(* IEC 61131-3 sources: Word/plc-course/05-boolean-logic-and-fbd/labs/solutions, 3 files *)

(* ---- 05-1-pump-permissive.st ---- *)
(* Lab 05-1: Transfer pump P-101 start permissive.
   Module 05 (Boolean logic and FBD). REFERENCE SOLUTION - try the lab yourself first.

   Everything here is combinational: every output depends only on the inputs
   of the present scan. There is no seal-in, latch or timer. *)

PROGRAM TransferPump
  VAR (* I/O - addresses follow the OpenPLC convention *)
    SuctionOpenLS AT %IX0.0 : BOOL;  (* Suction valve XV-100 open limit switch (ZSO-100): TRUE = fully open *)
    LSL101_NC     AT %IX0.1 : BOOL;  (* Tank low-level switch LSL-101, NC: TRUE = level above the switch (healthy) *)
    MotorFault    AT %IX0.2 : BOOL;  (* Motor protection relay fault contact, NO: TRUE = protection tripped *)
    ManualSel     AT %IX0.3 : BOOL;  (* MAN-OFF-AUTO selector, MAN contact *)
    AutoSel       AT %IX0.4 : BOOL;  (* MAN-OFF-AUTO selector, AUTO contact *)
    Demand        AT %IX0.5 : BOOL;  (* Auto demand from the process: TRUE = liquid wanted *)
    ManualRunCmd  AT %IX0.6 : BOOL;  (* Manual run command, maintained: TRUE = run *)
    Pump          AT %QX0.0 : BOOL;  (* P-101 motor starter: TRUE = run *)
    PermissiveOK  AT %QX0.1 : BOOL;  (* White "Ready" lamp: all start permissives healthy *)
    SelectorFault AT %QX0.2 : BOOL;  (* Both selector contacts made at once *)
  END_VAR
  VAR (* internal *)
    AutoMode   : BOOL;  (* selector cleanly in AUTO *)
    ManualMode : BOOL;  (* selector cleanly in MAN *)
    RunRequest : BOOL;  (* the active mode is asking for the pump *)
  END_VAR

  (* 1. Permissives. Each input is used in the sense that means "healthy":
        LSL101_NC is wired fail-safe and is already TRUE when healthy, so it is
        used as it is. MotorFault is TRUE when faulted, so it needs a NOT. *)
  PermissiveOK := SuctionOpenLS AND LSL101_NC AND NOT MotorFault;

  (* 2. Mode. A healthy three-position selector closes at most one contact.
        Both contacts at once is a fault, and it must not select any mode. *)
  SelectorFault := ManualSel AND AutoSel;
  AutoMode      := AutoSel AND NOT ManualSel;
  ManualMode    := ManualSel AND NOT AutoSel;

  (* 3. What the active mode asks for. The parentheses are not strictly needed
        (AND binds tighter than OR), but they show the intent at a glance. *)
  RunRequest := (AutoMode AND Demand) OR (ManualMode AND ManualRunCmd);

  (* 4. The permissives apply in every mode, so they go outside the OR. *)
  Pump := PermissiveOK AND RunRequest;
END_PROGRAM

CONFIGURATION Config0
  RESOURCE Res0 ON PLC
    TASK MainTask(INTERVAL := T#10ms, PRIORITY := 0);
    PROGRAM Inst0 WITH MainTask : TransferPump;
  END_RESOURCE
END_CONFIGURATION

(* ---- 05-2-two-out-of-three-vote.st ---- *)
(* Lab 05-2: Two-out-of-three (2oo3) high-pressure trip vote.
   Module 05 (Boolean logic and FBD). REFERENCE SOLUTION - try the lab yourself first.

   TRAINING EXERCISE ONLY. This shows the Boolean logic of voting. It is not a
   design for a real safety function: real trips run in a safety-rated system
   engineered to IEC 61511 / IEC 61508 (Module 20), and they latch until reset. *)

PROGRAM TripVote
  VAR (* I/O - addresses follow the OpenPLC convention *)
    PSHH_A_NC   AT %IX0.0 : BOOL;  (* PSHH-101A, NC: TRUE = pressure below trip setting (healthy) *)
    PSHH_B_NC   AT %IX0.1 : BOOL;  (* PSHH-101B, NC: as above *)
    PSHH_C_NC   AT %IX0.2 : BOOL;  (* PSHH-101C, NC: as above *)
    Trip        AT %QX0.0 : BOOL;  (* TRUE = at least two channels demand a trip *)
    SDVSolenoid AT %QX0.1 : BOOL;  (* SDV-100 solenoid: TRUE = energised, valve held open *)
    Discrepancy AT %QX0.2 : BOOL;  (* TRUE = the three channels do not all agree *)
    DiscA       AT %QX0.3 : BOOL;  (* TRUE = channel A disagrees with B and C *)
    DiscB       AT %QX0.4 : BOOL;  (* TRUE = channel B disagrees with A and C *)
    DiscC       AT %QX0.5 : BOOL;  (* TRUE = channel C disagrees with A and B *)
  END_VAR
  VAR (* internal: channel trip demands, TRUE = this channel says "trip" *)
    DemA : BOOL;
    DemB : BOOL;
    DemC : BOOL;
  END_VAR

  (* 1. Convert each fail-safe input into "this channel demands a trip".
        High pressure opens the contact, and so does a broken wire: both
        read FALSE, and both count as a demand. *)
  DemA := NOT PSHH_A_NC;
  DemB := NOT PSHH_B_NC;
  DemC := NOT PSHH_C_NC;

  (* 2. Majority vote: any two of the three. *)
  Trip := (DemA AND DemB) OR (DemB AND DemC) OR (DemA AND DemC);

  (* 3. De-energise to trip: the solenoid is powered only while there is no trip. *)
  SDVSolenoid := NOT Trip;

  (* 4. Which channel is the odd one out? A channel disagrees with the others
        when it differs from BOTH of them (which also means the other two agree). *)
  DiscA := (DemA XOR DemB) AND (DemA XOR DemC);
  DiscB := (DemB XOR DemA) AND (DemB XOR DemC);
  DiscC := (DemC XOR DemA) AND (DemC XOR DemB);

  (* 5. With three two-state channels, "not all equal" always means exactly
        one channel is the odd one out, so this is the same as
        (DemA XOR DemB) OR (DemB XOR DemC). *)
  Discrepancy := DiscA OR DiscB OR DiscC;
END_PROGRAM

CONFIGURATION Config0
  RESOURCE Res0 ON PLC
    TASK MainTask(INTERVAL := T#10ms, PRIORITY := 0);
    PROGRAM Inst0 WITH MainTask : TripVote;
  END_RESOURCE
END_CONFIGURATION

(* ---- 05-3-horn-truth-table.st ---- *)
(* Lab 05-3: From truth table to minimal logic - wet-well alarm horn.
   Module 05 (Boolean logic and FBD). REFERENCE SOLUTION - try the lab yourself first.

   K-map (rows HighLevel LowLevel, columns Pump1Run Pump2Run, Gray order):

                    P1 P2:  00   01   11   10
     H L = 00               0    0    0    0
     H L = 01               0    1    1    1
     H L = 11               1    1    1    1
     H L = 10               1    0    0    0

   Groups:  L.P2      quad  (rows 01, 11 x columns 01, 11)
            L.P1      quad  (rows 01, 11 x columns 11, 10)
            H.P1'.P2' pair  (rows 11, 10 x column 00)
   Every group is essential, so the minimal sum of products is unique:
     Horn = L.P1 + L.P2 + H.P1'.P2'     (3 terms, 7 literals)

   Reading the terms back as plant rules:
     L.P1, L.P2   a pump is running while the low-level float says "low":
                  the pump is about to run dry.
     H.P1'.P2'    high level and no pump running: the pumps have failed.
   Both floats "on" at once (a float fault) sounds the horn anyway: with no
   pump running the H term covers it, and with a pump running the L terms do,
   so no separate term is needed. *)

PROGRAM WetWellHorn
  VAR (* I/O - addresses follow the OpenPLC convention *)
    HighLevel AT %IX0.0 : BOOL;  (* High-level float relay: TRUE = level high *)
    LowLevel  AT %IX0.1 : BOOL;  (* Low-level float relay: TRUE = level low *)
    Pump1Run  AT %IX0.2 : BOOL;  (* Pump 1 running (contactor auxiliary contact) *)
    Pump2Run  AT %IX0.3 : BOOL;  (* Pump 2 running (contactor auxiliary contact) *)
    Horn      AT %QX0.0 : BOOL;  (* Wet-well alarm horn *)
  END_VAR

  Horn := (LowLevel AND Pump1Run)
       OR (LowLevel AND Pump2Run)
       OR (HighLevel AND NOT Pump1Run AND NOT Pump2Run);
END_PROGRAM

CONFIGURATION Config0
  RESOURCE Res0 ON PLC
    TASK MainTask(INTERVAL := T#10ms, PRIORITY := 0);
    PROGRAM Inst0 WITH MainTask : WetWellHorn;
  END_RESOURCE
END_CONFIGURATION
